PROGRAM prgHeizen
VAR
  // Modbus Hoval


  //Temperatursensor OG1 Büro (Shelly)
  fbOG1BueroTemperatur  : FB_ShellyHT_Udp:= (Start:= TRUE, Port:= 50001);
	OG1BueroTemperatur		: LREAL;			//{#lynus.ag#()}
	OG1BueroFeuchte    		: LREAL;			//{#lynus.ag#()}
	OG1BueroBatterie   		: LREAL;			//{#lynus.ag#()}


END_VAR

{region "Temperatursensor OG1 Büro (Shelly)"}
  fbOG1BueroTemperatur();

	OG1BueroTemperatur:= fbOG1BueroTemperatur.Temperatur;
	OG1BueroFeuchte   := fbOG1BueroTemperatur.Feuchte;
	OG1BueroBatterie  := fbOG1BueroTemperatur.Batterie;
{endregion}

END_PROGRAM

(* stored: Version 1.1.0.1, ProductVersion 3.1.4024.15
   POU prgHeizen: Id {92189520-e6a7-44cd-8fe5-f9273c6a4ce8}, SpecialFunc None *)
